// TwinCAT 3 PLC project Black_Jack_Practice
// ProgramVersion: 3.1.4023.0
// libraries:
//   Tc2_Standard, * (Beckhoff Automation GmbH)
//   Tc2_System, * (Beckhoff Automation GmbH)
//   Tc3_Module, * (Beckhoff Automation GmbH)
// project tree:
//   DUTs/ E_BlackJackVariation.TcDUT, E_SideBetChoice.TcDUT, ST_BasicStrategy.TcDUT, ST_BlackJackVariation.TcDUT, ST_GameAnalysis.TcDUT, ST_GamePlay.TcDUT, ST_GameSetup.TcDUT, ST_HardTotals.TcDUT, ST_HMI.TcDUT, ST_Messages.TcDUT, ST_PairSplitting.TcDUT, ST_Player.TcDUT, ST_PlayerHelp.TcDUT, ST_Dealer.TcDUT, ST_SideBetChoice.TcDUT, ST_SideBetInfo.TcDUT, ST_SoftTotals.TcDUT, ST_StepSequencer.TcDUT, ST_SurrenderHands.TcDUT, ST_Table_Info.TcDUT
//   GVLs/ GVL_Global.TcGVL
//   / PlcTask.TcTTO
//   POUs/ FB_Clear.TcPOU, FB_GamePlay.TcPOU, FB_GameSetup.TcPOU, FB_HMI.TcPOU, FB_MessageRecording.TcPOU, MAIN.TcPOU
// real-time tasks:
//   TASK PlcTask: cycle T#10ms, priority 20, ADS port 350

CONFIGURATION Black_Jack_Practice
    RESOURCE PLC ON TwinCAT3
        TASK PlcTask(INTERVAL := T#10ms, PRIORITY := 20);
        PROGRAM MAIN WITH PlcTask : MAIN;
    END_RESOURCE
END_CONFIGURATION

// ---- DUTs/E_BlackJackVariation.TcDUT
{attribute 'qualified_only'}
{attribute 'strict'}
TYPE E_BlackJackVariation :
(
	Idle				:= 0,
	Common_BlackJack 	:= 1,
	FreeBet_BlackJack	:= 2,
	Spanish21			:= 3
	
);
END_TYPE

// ---- DUTs/E_SideBetChoice.TcDUT
{attribute 'qualified_only'}
{attribute 'strict'}
TYPE E_SideBetChoice :
(
	BusterBlackjack := 0,
	Dealer16 := 1,
	LuckyLucky := 2,
	MatchtheDealer := 3
);
END_TYPE

// ---- DUTs/ST_BasicStrategy.TcDUT
TYPE ST_BasicStrategy :
STRUCT
	stHardTotals		:	ST_HardTotals;		//Hard Totals - Player has a total of 8 to 17
	stPairSplitting		:	ST_PairSplitting;	//Pair Splitting - Player receives two of the same card
	stSoftTotals		:	ST_SoftTotals;		//Soft Totals - Player has an A and  a 2-9
	stSurrenderHands	:	ST_SurrenderHands;	//Surrender Hands - Player has a total that is best to surrender
END_STRUCT
END_TYPE

// ---- DUTs/ST_BlackJackVariation.TcDUT
TYPE ST_BlackJackVariation :
STRUCT
	bCommonBlackJack	: BOOL; //Common Black Jack
	bFreeBetBlackJack	: BOOL;	//Free Bet Black Jack
	bSpanish21			: BOOL; //Spanish 21
END_STRUCT
END_TYPE

// ---- DUTs/ST_GameAnalysis.TcDUT
TYPE ST_GameAnalysis :
STRUCT
	aShoe				: ARRAY[0..999] OF STRING(255);	//Cards left in shoe to deal
	iCardsLeft			: DINT;							//Cards left to deal
	iCardsStartedWith	: DINT;							//Cards to deal at the start of the game
	iDecksStartedWith	: DINT;							//Decks that will be dealt
	rDecksLeft			: REAL;							//Decks left to deal
	
END_STRUCT
END_TYPE

// ---- DUTs/ST_GamePlay.TcDUT
TYPE ST_GamePlay :
STRUCT
	//Vars
	bClear					: BOOL;							//Clear all variables
 	bInitialStart			: BOOL;							//Initial start to the game		
	bReadyToStart			: BOOL;							//Game can now be started
	bStart					: BOOL;							//Start program
	bVariationSelected		: BOOL;							//Variation has been selected
	iStepNumber				: DINT;							//Game Play Sequence Step number
	iVariationSelection		: DINT;							//User selection for BlackJack variation
	
	//Structs
	sMessageType			: ST_Messages;					//Messages for feeback to player
	bStep					: ST_StepSequencer;  			//Game Play Sequence Step number trigger
	
	//Enums
	eBJVariation			: E_BlackJackVariation;			//BlackJack variation
END_STRUCT
END_TYPE

// ---- DUTs/ST_GameSetup.TcDUT
TYPE ST_GameSetup :
STRUCT
	//Vars
	bVariationSelected		: BOOL;							//Variation has been selected
	bSideBetChoice_One		: BOOL;							//First side bet picked
	bSideBetChoice_Two		: BOOL;							//Second side bet picked
	bBankRollComplete		: BOOL;							//Bank roll for each player has been inputed
	bGameSetupComplete		: BOOL;							//Game setup has been complete
	iStepNumber				: DINT;							//Game Play Sequence Step number
	iSeatsOpen				: DINT;							//Seats/hand left open
	sCards					: ARRAY[0..13] OF STRING(255);	//Array for card values in a deck
	sCardSuit				: ARRAY[0..3] OF STRING(255);	//Array of card suits in a deck
	
	//Structs
	stMessageType			: ST_Messages;					//Messages for feeback to player
	stStep					: ST_StepSequencer;  			//Game Play Sequence Step number trigger
	stPlayer				: ARRAY[1..6] OF ST_Player;
	stSideBetChoice			: ST_SideBetChoice;
END_STRUCT
END_TYPE

// ---- DUTs/ST_HardTotals.TcDUT
TYPE ST_HardTotals :
STRUCT
	//Player has a 8 or lower, always hit.
	//Player has a 9 and dealer showing a 3-6, double. Otherwise, hit.
	//Player has a 10 and dealer showing a 10 or A, stand. Otherwise, double.
	//Player has a 11, always double.
	//Player has a 12 and dealer showing a 4-6, stand. Otherwise, hit.
	//Player has a 13-16 and dealer showing a 2-6, stand. Otherwise, hit.
	//Player has a 17 or higher, always stand.
END_STRUCT
END_TYPE

// ---- DUTs/ST_HMI.TcDUT
TYPE ST_HMI :
STRUCT
	bClear				: BOOL; //Clear all arrays, variables
	bHMIRefresh			: BOOL; //Refresh HMI variables
	bOnline				: BOOL;	//HMI is online
	bStartHMIProgram	: BOOL;	//Start HMI program
	bUploadInfo			: BOOL; //Upload infomration on HMI
END_STRUCT
END_TYPE

// ---- DUTs/ST_Messages.TcDUT
TYPE ST_Messages :
STRUCT
	bErrorMessage				: BOOL;							//Error message has been displayed
	bFeedbackMessage			: BOOL;							//Feedback message has been displayed
	bInstructionMessage			: BOOL;							//Instruction message has been displayed
	bMessageToBeRecorded		: BOOL;							//Need to record message
	i							: DINT;							//Iterator
	sErrorMessage				: STRING(255);					//Error Instruction feedback to player
	sFeedbackMessage			: STRING(255);					//Feedback messages to player
	sInstructionMessage			: STRING(255);					//Instruction messages to player
	sErrorMessageHistory		: ARRAY[0..99] OF STRING(255);	//Error message history log
	sFeedbackMessageHistory		: ARRAY[0..99] OF STRING(255);	//Feedback message history
	sInstructionMessageHistory	: ARRAY[0..99] OF STRING(255);	//Instruction message history
	sRulesForGame				: ARRAY[0..99] OF STRING(255);	//Game rules for deviation
END_STRUCT
END_TYPE

// ---- DUTs/ST_PairSplitting.TcDUT
TYPE ST_PairSplitting :
STRUCT
	//Player has a pair of 2s or 3s and dealer showing a 2 or 3, split if allowed to double after split. Otherwise, don't split.
	//Player has a pair of 2s or 3s and dealer showing a 4-7, split. If dealer shows a 8 or higher don't split.
	//Player has a pair of 4s and dealer showing a 5 or 6, split if allowed to double after split. Otherwise, don't split.
	//Player has a pair of 5s, never split.
	//Player has a pair of 6s and dealer showing a 2, split if allowed to double after split. Otherwise, don't split.
	//Player has a pair of 6s and dealer showing a 3-6, split. Otherwise, don't split.
	//Player has a pair of 7s and dealer showing a 2-7, split. Otherwise, don't split.
	//Player has a pair of 8s, always split.
	//Player has a pair of 9s and dealer shows a 2-6, 8, or 9, split. Otherwise, don't split.
	//Player has a pair of 10s, never split.
	//Player has a pair of As, always split.
END_STRUCT
END_TYPE

// ---- DUTs/ST_Player.TcDUT
TYPE ST_Player :
STRUCT
	//Player hand
	sCard				: ARRAY[0..9] OF STRING(255); 	//Each card player has drawn
	sCardSuit			: ARRAY[0..9] OF STRING(255); 	//Each card's suit player has drawn	
	bBust				: BOOL;							//Player's has busted
	bSeatPlaying		: BOOL;							//Seat/hand is occupied to play
	bSeatNotPlaying		: BOOL;							//Seat/hand is not being occupied
	iHandTotal			: DINT;							//Player's hand total
	iNumberofCards		: DINT;							//Number of cards player has drawn
	iStartingBankRoll	: DINT;							//Player's starting bank roll
	iSeat				: DINT;							//Player's seat (1-6)
	sHand				: ARRAY[0..9] OF STRING(255);	//Player Hand
	rAvailableBalance	: REAL;							//Available balance player still has
	rBetAmount			: REAL;							//Amount player is betting
	rTotal				: REAL;							//Cash amount player is leaving with
	
END_STRUCT
END_TYPE

// ---- DUTs/ST_PlayerHelp.TcDUT
TYPE ST_PlayerHelp :
STRUCT
	stBasicStrategy	: ST_BasicStrategy; //Basic strategy for playing common Black Jack 
END_STRUCT
END_TYPE

// ---- DUTs/ST_Dealer.TcDUT
TYPE ST_Dealer :
STRUCT
	//Dealer hand
	sCard			:	ARRAY[0..9] OF STRING(255); 	//Each card dealer has drawn
	sCardSuit		:	ARRAY[0..9] OF STRING(255); 	//Each card's suit dealer has drawn	
	bBust			:	BOOL;							//Dealer has busted
	iHandTotal		:	DINT;							//Dealer's hand total
	iNumberofCards	:	DINT;							//Number of cards dealer has drawn
	sHand			: ARRAY[0..9] OF STRING(255);		//Dealer Hand
	
END_STRUCT
END_TYPE

// ---- DUTs/ST_SideBetChoice.TcDUT
TYPE ST_SideBetChoice :
STRUCT
	bBusterBlackjackSelected	: BOOL;			//Buster Blackjack was chosen
	bDealer16Selected			: BOOL;			//Dealer 16 was chosen
	bLuckyLuckySelected			: BOOL;			//Lucky Lucky was chosen
	bMatchtheDealerSelected		: BOOL;			//Match the dealer was chosen
	bPotofGoldSelected			: BOOL;			//Pot of Gold was chosen
	iFind						: INT;			//Variable keeping track of side bet selections
	sSideBetSelections			: STRING(255);	//Side Bet choices
	sSideBetSelectionsDecoded	: STRING(255);	//Side Bet choices decoded to find side bet selections
	iSideBet_One				: INT;  		//Side bet selection #1
	iSideBet_Two				: INT;  		//Side bet selection #2
	iSideBetSelections			: UINT;			//Side bet selections permissives
	
	//Structs
	stBusterBlackJack			: ST_SideBetInfo; //Buster Black Jack side bet
	stDealer16					: ST_SideBetInfo; //Dealer 16 side bet - dealer must got a 6 and 10 with first 2 cards
	stLuckyLucky				: ST_SideBetInfo; //Lucky Lucky side bet
	stMatchtheDealer			: ST_SideBetInfo; //Match the Dealer side bet
	stPotofGold					: ST_SideBetInfo; //Pot of Gold side bet (TBD)
	
	//Enums
	eSideBetChoice				: E_SideBetChoice;
END_STRUCT
END_TYPE

// ---- DUTs/ST_SideBetInfo.TcDUT
TYPE ST_SideBetInfo :
STRUCT
	aRules	: ARRAY[0..31] OF STRING(255); //Rules for side bet
	
END_STRUCT
END_TYPE

// ---- DUTs/ST_SoftTotals.TcDUT
TYPE ST_SoftTotals :
STRUCT
	//Player has a A,2 or A,3 and dealer showing a 5 or 6, double. Otherwise, hit.
	//Player has a A,4 or A,5 and dealer showing a 4, 5 or 6, double. Otherwise, hit.
	//Player has a A,6 and dealer showing a 3-6, double. Otherwise, hit.
	//Player has a A,7 and dealer showing a 2-6, double if allowed. If not, stand on a dealer 2-8 or hit on a dealer 9-10. 
	//Player has a A,8 and dealer showing a 6, double if allowed. If not, always stand on every hand.
	//Player has a A,9 always stand.
END_STRUCT
END_TYPE

// ---- DUTs/ST_StepSequencer.TcDUT
TYPE ST_StepSequencer :
STRUCT
	bStep					: ARRAY [0..63] OF BOOL;  		//Game Play Sequence Step number trigger
END_STRUCT
END_TYPE

// ---- DUTs/ST_SurrenderHands.TcDUT
TYPE ST_SurrenderHands :
STRUCT
	//Player has a 15 and dealer is showing a 10
	//Player has a 16 and dealer is showing a 9, 10 or A
END_STRUCT
END_TYPE

// ---- DUTs/ST_Table_Info.TcDUT
TYPE ST_Table_Info :
STRUCT
	bSideBets				:	BOOL; //Determines if side bets will be played.
	iInsuranceOdds			:	DINT; //Percentage or ratio that insurance will pay.
	iMinimumBet				:	DINT; //Minimum table bet that each player must put in if 
	iNumberofDecks			:	DINT; //Number of decks that will be dealt.
	iNumberofPlayers		:	DINT; //Number of players that will play (Max 6 players).
	rTableOdds				:	REAL; //Percentage or ratio that table deals for a Black Jack.
	
	//Structs
	stBlackJackVariation	:	ST_BlackJackVariation;	//Type of Black Jack variation to play.
	stSideBetChoice			:	ST_SideBetChoice;		//Side bets available to play.
	
	//Enums
	eBlackJackVariation		:	E_BlackJackVariation; 	//Type of Black Jack variation to play.
	
	
	
END_STRUCT
END_TYPE

// ---- GVLs/GVL_Global.TcGVL
{attribute 'qualified_only'}
VAR_GLOBAL
	//Vars
	bClear_Complete			: BOOL;							//Clear command complete
	bEndGame				: BOOL;							//Game has been ended.
	bGameInProgress			: BOOL;							//Game is running
	bGameIsPaused			: BOOL;							//Game is paused
    bInitialStart			: BOOL;							//Initial start to the game	- controlled by user	
	bReadyToStart			: BOOL;							//Game can now be started
	bStep					: ARRAY [0..63] OF BOOL;  		//Game Play Sequence Step number trigger
	bVariationSelected		: BOOL;							//Variation has been selected
	iStepNumber				: DINT;							//Game Play Sequence Step number
	iVariationSelection		: DINT;							//User selection for BlackJack variation
	sErrorInstruction		: STRING(255);					//Error Instruction feedack to player
	sSetupInstructions		: ARRAY[0..99] OF STRING(255);	//Set up instructions for game play
	sInstruction			: STRING(255);					//Instruction for player
	sCardNumbers			: ARRAY[0..12] OF STRING(255);  //Card numbers in a deck (2-10, J, K, Q, A)
	sCardSuit				: ARRAY[0..4] OF STRING(255);   //Card suits - 4 cards of each suit Clubs, Diamonds, Bishops, Hearts)	
	
	//Structs
	stDealer				: ST_Dealer;					//Dealer info
	stGamePlay				: ST_GamePlay;					//Game play vars
	stGameSetup				: ST_GameSetup;
	stHelp					: ST_PlayerHelp;				//Help for player to reference basic strategy for common blackjack
	stHMI					: ST_HMI;						//HMI variables
	stPlayer				: ARRAY[0..5] OF ST_Player;		//Player(s) info
	stTable					: ST_Table_Info;				//Black Jack table information
	stStepSequencer			: ST_StepSequencer;				//Sequencer
	
	//Enums
	eBJVariation			: E_BlackJackVariation;			//BlackJack variation
END_VAR

// ---- POUs/MAIN.TcPOU
PROGRAM MAIN
VAR
END_VAR

FB_GamePlay();

END_PROGRAM

// ---- POUs/FB_GamePlay.TcPOU
FUNCTION_BLOCK FB_GamePlay
VAR_INPUT
END_VAR
VAR_OUTPUT
END_VAR
VAR
END_VAR

// Decode sequencer step bits
MEMSET(ADR(GVL_Global.bStep), 0, SIZEOF(GVL_Global.bStep));
GVL_Global.bStep[GVL_Global.iStepNumber] := TRUE;

//States
// 0 = Idle - Game is waiting for user to start game
IF GVL_Global.bStep[0] THEN
	IF GVL_Global.stGamePlay.bClear THEN
		GVL_Global.iStepNumber := 1;
	END_IF
	
	IF GVL_Global.stGamePlay.bStart THEN
		GVL_Global.iStepNumber := 2;
	END_IF
	
// 1 = Clear - Clear all variables
ELSIF GVL_Global.bStep[1] THEN
	FB_Clear();
	IF GVL_Global.bClear_Complete THEN
		GVL_Global.stGamePlay.bClear := FALSE;
		GVL_Global.bClear_Complete := FALSE;
		GVL_Global.iStepNumber := 0;
	END_IF
	
// 2 = Game Set Up - Game to get set up to play
ELSIF GVL_Global.bStep[2] THEN
	IF GVL_Global.bReadyToStart THEN
		IF GVL_Global.bInitialStart THEN
			FB_GameSetup();
			IF GVL_Global.stGameSetup.bGameSetupComplete THEN
				GVL_Global.bInitialStart := FALSE;
				GVL_Global.bGameInProgress := TRUE;
				GVL_Global.iStepNumber := 3;
			END_IF
		ELSE
			IF GVL_Global.bGameInProgress THEN
				GVL_Global.iStepNumber := 3;
			ELSE
				GVL_Global.iStepNumber := 0;
			END_IF
		END_IF
	ELSE
		FB_Clear();
	END_IF
	
// 3 = Game Is Ongoing - Game is currently being played
ELSIF GVL_Global.bStep[3] THEN
	IF GVL_Global.bGameInProgress THEN
		;
	END_IF
	;
	
// 4 = Pause Game - Game is paused or people have left the table
ELSIF GVL_Global.bStep[4] THEN
	;
	
// 5 = End Game - Finish game and display results
ELSIF GVL_Global.bStep[5] THEN
	;
// 63-999 = Error State
ELSIF GVL_Global.bStep[63] THEN
	;
END_IF

END_FUNCTION_BLOCK

// ---- POUs/FB_Clear.TcPOU
FUNCTION_BLOCK FB_Clear
VAR_INPUT
END_VAR
VAR_OUTPUT
END_VAR
VAR
	i	: INT;
	j	: INT;
	k	: INT;
END_VAR

//Clear Player(s) Info
FOR k := 0 TO 5 DO
	GVl_Global.stPlayer[k].bBust := FALSE;
	GVL_Global.stPlayer[k].iHandTotal := 0;
	GVL_Global.stPlayer[k].iNumberofCards := 0;
	GVL_Global.stPlayer[k].rAvailableBalance := 0;
	GVL_Global.stPlayer[k].rBetAmount := 0;
	GVL_Global.stPlayer[k].rTotal := 0;
	GVL_Global.stPlayer[k].sHand[k] := '';
	IF k >= 5 THEN
		GVL_Global.stPlayer[k].sHand[6] := '';
		GVL_Global.stPlayer[k].sHand[7] := '';
		GVL_Global.stPlayer[k].sHand[8] := '';
		GVL_Global.stPlayer[k].sHand[9] := '';
	END_IF
END_FOR

FOR i := 0 TO 9 DO
	GVL_Global.stPlayer[i].sCard[i] := '';
	GVL_Global.stPlayer[i].sCardSuit[i] := '';
	GVL_Global.stDealer.sCard[i] := '';
	GVL_Global.stDealer.sCardSuit[i] := '';
END_FOR

//Clear Dealer Info
GVl_Global.stDealer.bBust := FALSE;
GVL_Global.stDealer.iHandTotal := 0;
GVL_Global.stDealer.iNumberofCards := 0;
FOR j := 0 TO 9 DO
	GVL_Global.stDealer.sHand[j] := '';	
END_FOR

//Clear Table Info
GVL_Global.stTable.bSideBets := FALSE;
GVL_Global.stTable.iInsuranceOdds := 0;
GVL_Global.stTable.iMinimumBet := 0;
GVL_Global.stTable.iNumberofDecks := 0;
GVL_Global.stTable.iNumberofPlayers := 0;
GVL_Global.stTable.rTableOdds := 0;

GVL_Global.bClear_Complete := TRUE;
GVL_Global.bReadyToStart := TRUE;

END_FUNCTION_BLOCK

// ---- POUs/FB_GameSetup.TcPOU
FUNCTION_BLOCK FB_GameSetup
VAR_INPUT
END_VAR
VAR_OUTPUT
END_VAR
VAR
	i	: DINT;
	j	: DINT;
	k	: DINT;
	m	: INT;
END_VAR

// Decode sequencer step bits
MEMSET(ADR(GVL_Global.bStep), 0, SIZEOF(GVL_Global.bStep));
GVL_Global.stGameSetup.stStep[GVL_Global.stGameSetup.iStepNumber] := TRUE;

//Choose blackjack variation: 1 - Common BlackJack, 2 - Free Bet BlackJack, 3 - Spanish 21
IF GVL_Global.eBJVariation.Idle = GVL_Global.iVariationSelection THEN
	//Wait for user to select a BlackJack variation
	GVL_Global.sInstruction := 'Please choose a blackjack variation to play.';
END_IF

IF GVL_Global.iVariationSelection >= 1 AND GVL_Global.iVariationSelection <= 3 THEN
	//Set up initial information regarding card, card suit, and deck information
	FOR m := 0 TO 9 DO
		GVL_Global.stGameSetup.sCards[m] := INT_TO_STRING(m+2);
	END_FOR
	GVL_Global.stGameSetup.sCards[10] := 'J';
	GVL_Global.stGameSetup.sCards[11] := 'Q';
	GVL_Global.stGameSetup.sCards[12] := 'K';
	GVL_Global.stGameSetup.sCards[13] := 'A';
	
	GVL_Global.stGameSetup.sCardSuit[0] := 'Clubs';
	GVL_Global.stGameSetup.sCardSuit[1] := 'Diamonds';
	GVL_Global.stGameSetup.sCardSuit[2] := 'Bishops';
	GVL_Global.stGameSetup.sCardSuit[3] := 'Hearts';
	GVL_Global.stGameSetup.iStepNumber := 2;
ELSE
	GVL_Global.stGameSetup.iStepNumber := 0;
END_IF

//GVL_Global.sInstruction := 'Please choose a blackjack variation to play.';
//IF GVL_Global.iVariationSelection >=1 AND GVL_Global.iVariationSelection <= 3 THEN
//	GVL_Global.stGameSetup.iStepNumber := 2;
//ELSE
//	GVL_Global.stGameSetup.iStepNumber := 0;
//END_IF

//Error State
IF GVL_Global.stGameSetup.stStep.bStep[0] THEN
	//False entry was entered
	GVL_Global.stGamePlay.sMessageType.sErrorMessage := 'You entered a wrong variation input. Please try again.';
	GVL_Global.stGamePlay.bVariationSelected := FALSE;
	GVL_Global.stGamePlay.iVariationSelection := 0;
END_IF


//Idle State
IF GVL_Global.stGameSetup.stStep.bStep[1] THEN
	GVL_Global.stGamePlay.sMessageType.sErrorMessage := 'Game is ongoing.';
	IF GVL_Global.stGamePlay.bReadyToStart AND GVL_Global.stGameSetup.bBankRollComplete THEN
		GVL_Global.stGamePlay.iStepNumber := 1;
	ELSE
		GVL_Global.stGamePlay.iStepNumber := 0;
	END_IF
END_IF

//Blackjack Deviation Selection
IF GVL_Global.stGameSetup.stStep.bStep[2] THEN
	IF GVL_Global.eBJVariation.Common_BlackJack = GVL_Global.iVariationSelection THEN
		//Common Blackjack was selected
		GVL_Global.stGameSetup.stMessageType.sInstructionMessage := 'Variation selected: Common Blackjack.';
	ELSIF GVL_Global.eBJVariation.FreeBet_BlackJack = GVL_Global.iVariationSelection THEN
		GVL_Global.stGameSetup.stMessageType.sInstructionMessage := 'Variation selected: Free Bet Blackjack.';
	ELSIF GVL_Global.eBJVariation.Spanish21 = GVL_Global.iVariationSelection THEN
		GVL_Global.stGameSetup.stMessageType.sInstructionMessage := 'Variation selected: Spanish 21.';
	END_IF
	GVL_Global.stGameSetup.iStepNumber := 3;
END_IF

//Choose 2 sidebets: 1 - Buster BlackJack, 2 - Dealer 16, 3 - Lucky Lucky, 4 - Match the Dealer, 5 - Pot of Gold (TBD)
//Side Bets Selection
IF GVL_Global.stGameSetup.stStep.bStep[3] THEN
	GVL_Global.stGameSetup.stMessageType.sRulesForGame[0] := 'Choose two (2) side bets: 1 - Buster BlackJack, 2 - Dealer 16, 3 - Lucky Lucky, 4 - Match the Dealer, 5 - Pot of Gold';
	GVL_Global.stGameSetup.stMessageType.sInstructionMessage[1] := 'Enter in text box labeled -> Side Bets To Play';
	GVL_Global.stGameSetup.stMessageType.sInstructionMessage[2] := 'Choose two (2) side bets: 1 - Buster BlackJack, 2 - Dealer 16, 3 - Lucky Lucky, 4 - Match the Dealer, 5 - Pot of Gold';
	GVL_Global.stGameSetup.stMessageType.sInstructionMessage := 'Enter in the following prompt: #,#';
	//Side Bet Choices Decoded
	GVL_Global.stGameSetup.stSideBetChoice.iFind := FIND(',',GVL_Global.stGameSetup.stSideBetChoice.sSideBetSelections);
	GVL_Global.stGameSetup.stSideBetChoice.iSideBet_One := STRING_TO_INT(LEFT(GVL_Global.stGameSetup.stSideBetChoice.sSideBetSelections,GVL_Global.stGameSetup.stSideBetChoice.iFind-1));
	GVL_Global.stGameSetup.stSideBetChoice.iSideBet_Two := STRING_TO_INT(RIGHT(GVL_Global.stGameSetup.stSideBetChoice.sSideBetSelections,GVL_Global.stGameSetup.stSideBetChoice.iFind+1));
	//Side bet #1 chosen
	IF GVL_Global.stGameSetup.stSideBetChoice.iSideBet_One = GVL_Global.stGameSetup.stSideBetChoice.eSideBetChoice.BusterBlackjack THEN
		GVL_Global.stGameSetup.stSideBetChoice.bBusterBlackjackSelected := TRUE;
		//GVL_Global.stGameSetup.sSideBetChoice.iSideBetSelections.0 := TRUE;
	ELSIF GVL_Global.stGameSetup.stSideBetChoice.iSideBet_One = GVL_Global.stGameSetup.stSideBetChoice.eSideBetChoice.Dealer16 THEN
		GVL_Global.stGameSetup.stSideBetChoice.bDealer16Selected := TRUE;
		//GVL_Global.stGameSetup.sSideBetChoice.iSideBetSelections.1 := TRUE;
	ELSIF GVL_Global.stGameSetup.stSideBetChoice.iSideBet_One = GVL_Global.stGameSetup.stSideBetChoice.eSideBetChoice.LuckyLucky THEN
		GVL_Global.stGameSetup.stSideBetChoice.bLuckyLuckySelected := TRUE;
		//GVL_Global.stGameSetup.sSideBetChoice.iSideBetSelections.2 := TRUE;
	ELSIF GVL_Global.stGameSetup.stSideBetChoice.iSideBet_One = GVL_Global.stGameSetup.stSideBetChoice.eSideBetChoice.MatchtheDealer THEN
		GVL_Global.stGameSetup.stSideBetChoice.bMatchtheDealerSelected := TRUE;
	END_IF
	//Side bet #2 chosen
	IF GVL_Global.stGameSetup.stSideBetChoice.iSideBet_Two = GVL_Global.stGameSetup.stSideBetChoice.eSideBetChoice.BusterBlackjack THEN
		GVL_Global.stGameSetup.stSideBetChoice.bBusterBlackjackSelected := TRUE;
	ELSIF GVL_Global.stGameSetup.stSideBetChoice.iSideBet_Two = GVL_Global.stGameSetup.stSideBetChoice.eSideBetChoice.Dealer16 THEN
		GVL_Global.stGameSetup.stSideBetChoice.bDealer16Selected := TRUE;
	ELSIF GVL_Global.stGameSetup.stSideBetChoice.iSideBet_Two = GVL_Global.stGameSetup.stSideBetChoice.eSideBetChoice.LuckyLucky THEN
		GVL_Global.stGameSetup.stSideBetChoice.bLuckyLuckySelected := TRUE;
	ELSIF GVL_Global.stGameSetup.stSideBetChoice.iSideBet_Two = GVL_Global.stGameSetup.stSideBetChoice.eSideBetChoice.MatchtheDealer THEN
		GVL_Global.stGameSetup.stSideBetChoice.bMatchtheDealerSelected := TRUE;
	END_IF
	
	IF GVL_Global.stGameSetup.stSideBetChoice.iSideBet_One <> 0 AND GVL_Global.stGameSetup.stSideBetChoice.iSideBet_Two <> 0 THEN
		GVL_Global.stGameSetup.iStepNumber := 4;
	END_IF
END_IF

//Input number of players/hands to be dealt. Max of 6.
IF GVL_Global.stGameSetup.stStep.bStep[4] THEN
	GVL_Global.stGamePlay.sMessageType.sInstructionMessage := 'Please enter number of players/hands going to play';
	IF GVL_Global.stTable.iNumberofPlayers >= 1 AND GVL_Global.stTable.iNumberofPlayers <= 6 THEN
		//GVL_Global.stTable.iNumberofPlayers;
		FOR i := 1 TO GVL_Global.stTable.iNumberofPlayers DO
			GVL_Global.stGameSetup.stPlayer[i].bSeatPlaying := TRUE;	
		END_FOR
		//GVL_Global.stGameSetup.iSeatsOpen := GVL_Global.stTable.iNumberofPlayers + 1;
		GVL_Global.stGamePlay.iStepNumber := 5;
	ELSE
		//Number of players entered is invalid.
		GVL_Global.stGameSetup.stMessageType.sErrorMessage := 'Entered invalid number of players. Please try again.';
	END_IF
	//
//GVL_Global.stGamePlay.iStepNumber := 3;
END_IF

//Input number of decks to be dealt.
IF GVL_Global.stGameSetup.stStep.bStep[5] THEN
	GVL_Global.stGamePlay.sMessageType.sInstructionMessage := 'Please enter number of decks to deal (1-6)';
	IF GVL_Global.stTable.iNumberofDecks >= 1 AND GVL_Global.stTable.iNumberofDecks <= 6 THEN
		GVL_Global.stGamePlay.sMessageType.sInstructionMessage := CONCAT('Dealer will deal a total of ',DINT_TO_STRING(GVL_Global.stTable.iNumberofDecks));
		GVL_Global.stGamePlay.iStepNumber := 6;
	ELSE
		//Number of decks entered is invalid.
		GVL_Global.stGameSetup.stMessageType.sErrorMessage := 'Entered invalid number of decks. Please try again.';
	END_IF
END_IF

//Input table minimum bet.
IF GVL_Global.stGameSetup.stStep.bStep[6] THEN
	GVL_Global.stGamePlay.sMessageType.sInstructionMessage := 'Please enter the minimum bet to play.';
	IF GVL_Global.stTable.iMinimumBet >= 5 THEN
		GVL_Global.stGamePlay.sMessageType.sInstructionMessage := CONCAT('Minimum table bet is ',DINT_TO_STRING(GVL_Global.stTable.iMinimumBet));
		GVL_Global.stGamePlay.iStepNumber := 7;
	ELSE
		//Number of decks entered is invalid.
		GVL_Global.stGameSetup.stMessageType.sErrorMessage := 'Entered an invalid table bet. Please try again.';
	END_IF
END_IF

//Input table max bet. - May not use - TBD
IF GVL_Global.stGameSetup.stStep.bStep[7] THEN
	GVL_Global.stGamePlay.iStepNumber := 8;
END_IF

//Set up players/seats who are playing.
IF GVL_Global.stGameSetup.stStep.bStep[8] THEN
	FOR j := 1 TO GVL_Global.stTable.iNumberofPlayers DO
		GVL_Global.stGameSetup.stPlayer[j].iSeat := j;
	END_FOR
	GVL_Global.stGamePlay.iStepNumber := 9;
END_IF

//Input starting bank roll.
IF GVL_Global.stGameSetup.stStep.bStep[9] THEN
	GVL_Global.stGamePlay.sMessageType.sInstructionMessage := 'Please enter bankroll for each player.';
	IF GVL_Global.stGameSetup.bBankRollComplete THEN
		GVL_Global.stGamePlay.sMessageType := 'Details for chips: Reds - 5, Whites - 25, Blues - 100, Greens - 500, Blacks - 1 or 1000';
		GVL_Global.stGamePlay.iStepNumber := 10;
	END_IF
END_IF

//Chips given: Reds - $5, Whites - $25, Blues - $100, Greens - $500, Blacks - $1  

//Finalize Game Setup
IF GVL_Global.stGameSetup.stStep.bStep[10] THEN
	GVL_Global.stGamePlay.sMessageType.sInstructionMessage := 'Ready to start the game?';
	IF GVL_Global.stGamePlay.bReadyToStart THEN
		GVL_Global.stGameSetup.bGameSetupComplete := TRUE;
		GVL_Global.stGamePlay.iStepNumber := 1;
	END_IF
END_IF

END_FUNCTION_BLOCK

// ---- POUs/FB_HMI.TcPOU
FUNCTION_BLOCK FB_HMI
VAR_INPUT
END_VAR
VAR_OUTPUT
END_VAR
VAR
END_VAR

END_FUNCTION_BLOCK

// ---- POUs/FB_MessageRecording.TcPOU
FUNCTION_BLOCK FB_MessageRecording
VAR_INPUT
END_VAR
VAR_OUTPUT
END_VAR
VAR
END_VAR

IF GVL_Global.stGamePlay.sMessageType.bMessageToBeRecorded THEN
	IF GVL_Global.stGamePlay.sMessageType.bErrorMessage THEN
		;
	ELSIF GVL_Global.stGamePlay.sMessageType.bFeedbackMessage THEN
		;
	ELSIF GVL_Global.stGamePlay.sMessageType.bInstructionMessage THEN
		;
	END_IF
END_IF

END_FUNCTION_BLOCK
